Universal Robots PolyScope program: mirror-me.urp

Program mirror-me (installation=default directory=/programs createdIn=3.2.19275 lastSavedIn=5.19.0 robotSerialNumber=20245203260)
Calibrated DH parameters: a=[0.00002, -0.297909, -0.550376, -0.000026, 0.000029, 0]; d=[0.180392, 372.242289, -404.966968, 32.898661, 0.119952, 0.115576]; alpha=[1.570137, -0.001437, 0.004676, 1.569919, -1.569683, 0]; deltaTheta=[0, -1.062765, 0.791609, 0.271161, 0, 0]
InitVariablesNode
BeforeStart
  home_pose := p[0.05,-0.55,1.1,0,0,0]
  last_good_joint := [0,0,0,0,0,0]
  Script: last_good_joint = get_inverse_kin(home_pose)
  move_pose := home_pose
  Script: write_output_boolean_register(64,  False )
  Wait Sleep waitTime=0.1
  mode := 0
  j := [move_pose[0], move_pose[1], move_pose[2], move_pose[2], move_pose[4], move_pose[5],0]
  joints := [0,0,0,0,0,0]
  current_speed := 0.0
Robot Program (runOnlyOnce=false)
  Script: write_output_boolean_register(64, False)
  Script: mode = read_input_integer_register(0)
  Loop While (checkContinuously=false) expression=mode ≤ 4
    Loop While (checkContinuously=false) expression=mode ≟ 3
      Script: joints = get_inverse_kin(home_pose)
      Script: servoj(joints, t=0.02, lookahead_time=0.5, gain=0.2)
      Script: write_output_boolean_register(64, True )
      Script: mode = read_input_integer_register(0)
      Script: sync()
    Loop While (checkContinuously=false) expression=mode ≟ 4
      If current_speed < 1.0
        Script: current_speed = current_speed + 0.02
      Script: move_pose = p[j[0],j[1],j[2],0,0,0]
      Script: tool_pose = p[0,0,0,0,0,j[6]]
      Script: tool_pose = pose_trans(tool_pose, p[0,0,0.058,0,0,0])
      Script: tool_pose = pose_trans(tool_pose, p[0,0,0,j[3],j[4],j[5]])
      SuppressedNode
        Script: tool_pose = pose_add(tool_pose, p[0,0,0,0,j[4],0])
      SuppressedNode
        Script: tool_pose = pose_add(tool_pose, p[0,0,0,j[3],0,0])
      Script: move_pose = pose_trans(move_pose, tool_pose)
      If get_inverse_kin_has_solution(move_pose) and is_within_safety_limits(move_pose)
        Script file /programs/pose_limit.script
          | joints = get_inverse_kin(move_pose)
          | current_joints = get_actual_joint_positions()
          | max_change = [0.6, 0.35, 0.35, 0.45, 0.5, 0.5]
          | j_max = [3.05,-1.0472,2.44346,-0.174533,2.44346,3.14159]
          | j_min = [-1.48353,-2.61799,0.261799,-2.26893,0.872665,-3.14159]
          | 
          | s_off = 0.1
          | 
          | max_change = max_change * current_speed
          | 
          | NumChecks=6
          | 
          | joints_diff = joints - current_joints
          | Count=0
          | while Count < NumChecks:
          | 	if joints_diff[Count] > max_change[Count]:
          | 		joints[Count] = current_joints[Count] + max_change[Count]
          | 	end
          | 	if joints_diff[Count] < -max_change[Count]:
          | 		joints[Count] = current_joints[Count] - max_change[Count]
          | 	end
          | 	Count=Count+1
          | end
          | Count=0
          | while Count < NumChecks:
          | 	if joints[Count]  + s_off  > j_max[Count]:
          | 		textmsg("limit+ ", Count)
          | 		joints[Count] = j_max[Count] - s_off
          | 
          | 		textmsg("res ", joints[Count])
          | 	end
          | 	if joints[Count]  - s_off  < j_min[Count]:
          | 		textmsg("limit- ", Count)
          | 		joints[Count] = j_min[Count] + s_off
          | 		textmsg("res ", joints[Count])
          | 	end
          | 	Count = Count +1
          | end
        If is_within_safety_limits(joints)
          last_good_joint := joints
      Else 
        Script: current_speed = 0.0
      Script: servoj(last_good_joint, t=0.02, lookahead_time=0.1, gain=300)
      Script: write_output_boolean_register(64, True )
      Script: mode = read_input_integer_register(0)
      Script: sync()
    Script: mode = read_input_integer_register(0)
    Script: write_output_boolean_register(64, False)
    Script: sync()
Thread Thread_1 (runOnlyOnce=false)
  Loop Forever
    tmp := [0,0,0,0,0,0,0]
    Script: tmp[0] = read_input_float_register(0)
    Script: tmp[1] = read_input_float_register(1)
    Script: tmp[2] = read_input_float_register(2)
    Script: tmp[3] = read_input_float_register(3)
    Script: tmp[4] = read_input_float_register(4)
    Script: tmp[5] = read_input_float_register(5)
    Script: tmp[6] = read_input_float_register(6)
    j := tmp
    Script: sync()
